{attribute 'TcGenerated'}
// This function has been automatically generated from the project information.
VAR_GLOBAL CONSTANT
	{attribute 'const_non_replaced'}
	{attribute 'linkalways'}
	stLibVersion_Automation_components_gip : ST_LibVersion := (iMajor := 1, iMinor := 0, iBuild := 0, iRevision := 0, sVersion := '1.0.0');
END_VAR

(* stored: Version 1.1.0.1, ProductVersion 3.1.4020.6
   GVL Global_Version: Id {46304699-f3af-462e-bb5d-92b58a0a77c1} *)
